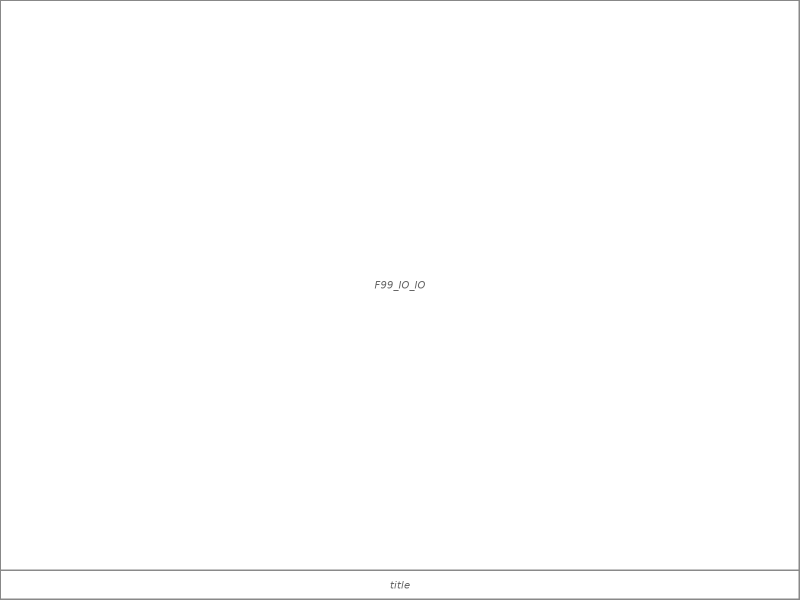
VISUALIZATION F99_Monitor  // 800x600
    Frame (0,570 800x30)
        shows title()
    TabControl (0,0 800x570)
        shows F99_IO_IO()
        shows F99_IO_IO_1()
        shows F99_IO_IO_2()
        shows F99_IO_ETHERCAT()
        shows F99_IO_SYSINFO()
        [3]: TabTitle=EtherCAT
        [4]: TabTitle=SysInfo
END_VISUALIZATION

(* stored: Version 1.1.0.1, ProductVersion 3.1.4024.11
   Visu F99_Monitor: Id {4c2085a0-04f4-4932-96b1-5bda1f310681} *)
